# EPICS autosave request: iocBoot/iocLabJack_T7Pro/auto_settings.req
file "LabJack_T7_settings.req", P=$(P)
